% RSLogix 500 project I2P JOB 14 - ANDREW_BAK032.RSS, saved by version 10.00.00.00 %
PROJECT "ML03A"    % processor: Bul.1763 MicroLogix 1100 Series B %

PROGRAM FILES
  LAD 2   12 rungs

DATA FILES
  O0 OUTPUT  4 elements
  I1 INPUT  6 elements
  S2 STATUS  66 elements
  B3 BINARY  1 elements
  T4 TIMER  1 elements
  C5 COUNTER  1 elements
  R6 CONTROL  1 elements
  N7 INTEGER  1 elements
  F8 FLOAT  1 elements

LADDER 2
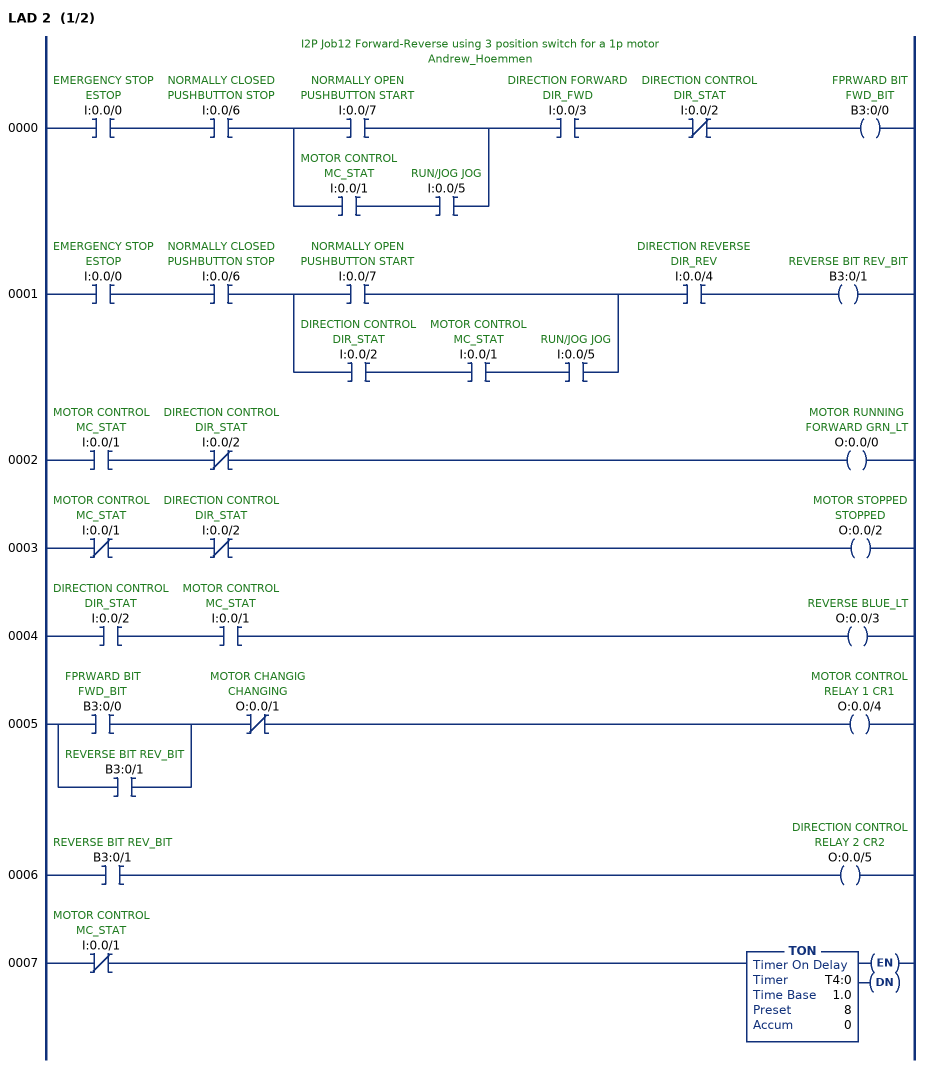
% Rung: 0 %
% I2P Job12 Forward-Reverse using 3 position switch for a 1p motor
% Andrew_Hoemmen %
SOR XIC I:0.0/0 XIC I:0.0/6 BST XIC I:0.0/7 NXB XIC I:0.0/1 XIC I:0.0/5 BND XIC I:0.0/3 XIO I:0.0/2 OTE B3:0/0 EOR
%   I:0.0/0  ESTOP  "EMERGENCY STOP" %
%   I:0.0/6  STOP  "NORMALLY CLOSED PUSHBUTTON" %
%   I:0.0/7  START  "NORMALLY OPEN PUSHBUTTON" %
%   I:0.0/1  MC_STAT  "MOTOR CONTROL" %
%   I:0.0/5  JOG  "RUN/JOG" %
%   I:0.0/3  DIR_FWD  "DIRECTION FORWARD" %
%   I:0.0/2  DIR_STAT  "DIRECTION CONTROL" %
%   B3:0/0  FWD_BIT  "FPRWARD BIT" %
% Rung: 1 %
SOR XIC I:0.0/0 XIC I:0.0/6 BST XIC I:0.0/7 NXB XIC I:0.0/2 XIC I:0.0/1 XIC I:0.0/5 BND XIC I:0.0/4 OTE B3:0/1 EOR
%   I:0.0/0  ESTOP  "EMERGENCY STOP" %
%   I:0.0/6  STOP  "NORMALLY CLOSED PUSHBUTTON" %
%   I:0.0/7  START  "NORMALLY OPEN PUSHBUTTON" %
%   I:0.0/2  DIR_STAT  "DIRECTION CONTROL" %
%   I:0.0/1  MC_STAT  "MOTOR CONTROL" %
%   I:0.0/5  JOG  "RUN/JOG" %
%   I:0.0/4  DIR_REV  "DIRECTION REVERSE" %
%   B3:0/1  REV_BIT  "REVERSE BIT" %
% Rung: 2 %
SOR XIC I:0.0/1 XIO I:0.0/2 OTE O:0.0/0 EOR
%   I:0.0/1  MC_STAT  "MOTOR CONTROL" %
%   I:0.0/2  DIR_STAT  "DIRECTION CONTROL" %
%   O:0.0/0  GRN_LT  "MOTOR RUNNING FORWARD" %
% Rung: 3 %
SOR XIO I:0.0/1 XIO I:0.0/2 OTE O:0.0/2 EOR
%   I:0.0/1  MC_STAT  "MOTOR CONTROL" %
%   I:0.0/2  DIR_STAT  "DIRECTION CONTROL" %
%   O:0.0/2  STOPPED  "MOTOR STOPPED" %
% Rung: 4 %
SOR XIC I:0.0/2 XIC I:0.0/1 OTE O:0.0/3 EOR
%   I:0.0/2  DIR_STAT  "DIRECTION CONTROL" %
%   I:0.0/1  MC_STAT  "MOTOR CONTROL" %
%   O:0.0/3  BLUE_LT  "REVERSE" %
% Rung: 5 %
SOR BST XIC B3:0/0 NXB XIC B3:0/1 BND XIO O:0.0/1 OTE O:0.0/4 EOR
%   B3:0/0  FWD_BIT  "FPRWARD BIT" %
%   B3:0/1  REV_BIT  "REVERSE BIT" %
%   O:0.0/1  CHANGING  "MOTOR CHANGIG" %
%   O:0.0/4  CR1  "MOTOR CONTROL RELAY 1" %
% Rung: 6 %
SOR XIC B3:0/1 OTE O:0.0/5 EOR
%   B3:0/1  REV_BIT  "REVERSE BIT" %
%   O:0.0/5  CR2  "DIRECTION CONTROL RELAY 2" %
% Rung: 7 %
SOR XIO I:0.0/1 TON T4:0 1.0 8 0 EOR
%   I:0.0/1  MC_STAT  "MOTOR CONTROL" %

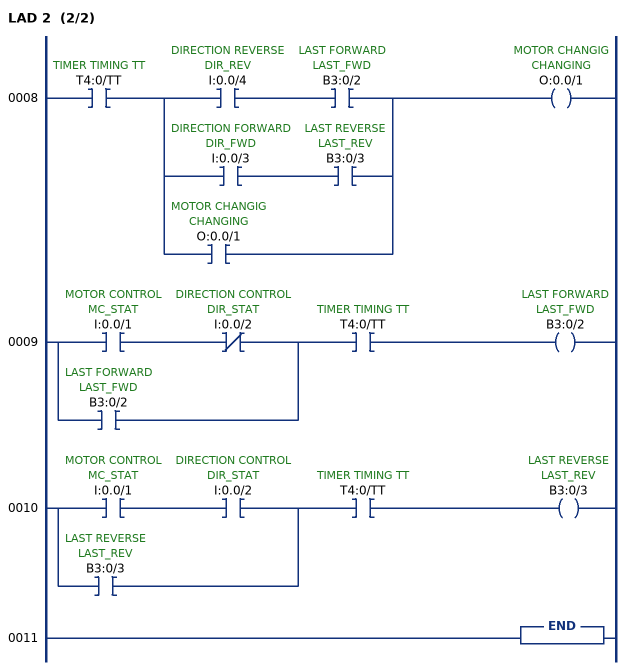
% Rung: 8 %
SOR XIC T4:0/TT BST XIC I:0.0/4 XIC B3:0/2 NXB BST XIC I:0.0/3 XIC B3:0/3 NXB XIC O:0.0/1 BND BND OTE O:0.0/1 EOR
%   T4:0/TT  TT  "TIMER TIMING" %
%   I:0.0/4  DIR_REV  "DIRECTION REVERSE" %
%   B3:0/2  LAST_FWD  "LAST FORWARD" %
%   I:0.0/3  DIR_FWD  "DIRECTION FORWARD" %
%   B3:0/3  LAST_REV  "LAST REVERSE" %
%   O:0.0/1  CHANGING  "MOTOR CHANGIG" %
% Rung: 9 %
SOR BST XIC I:0.0/1 XIO I:0.0/2 NXB XIC B3:0/2 BND XIC T4:0/TT OTE B3:0/2 EOR
%   I:0.0/1  MC_STAT  "MOTOR CONTROL" %
%   I:0.0/2  DIR_STAT  "DIRECTION CONTROL" %
%   B3:0/2  LAST_FWD  "LAST FORWARD" %
%   T4:0/TT  TT  "TIMER TIMING" %
% Rung: 10 %
SOR BST XIC I:0.0/1 XIC I:0.0/2 NXB XIC B3:0/3 BND XIC T4:0/TT OTE B3:0/3 EOR
%   I:0.0/1  MC_STAT  "MOTOR CONTROL" %
%   I:0.0/2  DIR_STAT  "DIRECTION CONTROL" %
%   B3:0/3  LAST_REV  "LAST REVERSE" %
%   T4:0/TT  TT  "TIMER TIMING" %
% Rung: 11 %
SOR END EOR

OTHER DOCUMENTED ADDRESSES
  I:0.0/8  PB3  "NORMALLY OPEN PUSHBUTTON"

DATA TABLE (non-zero values as saved)
DATA T4
% .PRE .ACC %
% T4:0 % 8 0
